FUNCTION_BLOCK Necessidade_2_Equipamentos_HMI (* Service Interface Function Block Type *)
  (* Standard: 61499-2 *)
  (* Version 0.0, 25/02/2026, template *)
  PACKAGE Hidryco.HidrycoLib;
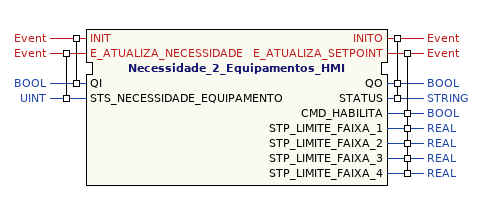
  EVENT_INPUT
    INIT WITH QI;
    E_ATUALIZA_NECESSIDADE WITH STS_NECESSIDADE_EQUIPAMENTO;
  END_EVENT
  EVENT_OUTPUT
    INITO WITH QO, STATUS;
    E_ATUALIZA_SETPOINT WITH STP_LIMITE_FAIXA_1, STP_LIMITE_FAIXA_2, STP_LIMITE_FAIXA_3, STP_LIMITE_FAIXA_4, CMD_HABILITA;
  END_EVENT
  VAR_INPUT
    QI : BOOL;
    STS_NECESSIDADE_EQUIPAMENTO : UINT;
  END_VAR
  VAR_OUTPUT
    QO : BOOL; (* Event Output Qualifier *)
    STATUS : STRING; (* Service Status *)
    CMD_HABILITA : BOOL;
    STP_LIMITE_FAIXA_1 : REAL;
    STP_LIMITE_FAIXA_2 : REAL;
    STP_LIMITE_FAIXA_3 : REAL;
    STP_LIMITE_FAIXA_4 : REAL;
  END_VAR
  SERVICE /
    SEQUENCE 
    END_SEQUENCE
  END_SERVICE
END_FUNCTION_BLOCK
